(* IEC 61131-3 sources: volt/packages/volt-lsp-iec/test-corpus/lenze-mid/Device/Plc Logic/Application/Library Manager/L_MC4P_RoboticHandling (part 4) *)

(* ---- L_MC4P_TEMPLATE_FORAG.pou ---- *)
FUNCTION_BLOCK L_MC4P_TEMPLATE_FORAG
VAR
	XERROROLD : BOOL;
	WERRORIDOLD : WORD;
	XDISABLEERRORRESET : BOOL;
	XDISABLEERRORLOGGING : BOOL;
	DWERRORITFID : DWORD;
	PFBBASEAXESGROUP : POINTER TO AXES_GROUP_REF;
	PSINSTANCESTR : POINTER TO STRING;
	DISABLEERRORLOGGING : BOOL;
	DISABLEERRORRESET : BOOL;
END_VAR
END_FUNCTION_BLOCK

METHOD SETINCTANCEINFO
VAR_INPUT
	PSINSTANCENAME : POINTER TO STRING;
	ERRORITFID : DWORD;
END_VAR
END_METHOD

METHOD SETINSTANCEINFOANDAXISPOINTER
VAR_INPUT
	PAXESGROUP : POINTER TO AXES_GROUP_REF;
	PSNAME : POINTER TO STRING;
END_VAR
END_METHOD

METHOD UPDATEAXISPOINTER
VAR_INPUT
	PAXESGROUP : POINTER TO AXES_GROUP_REF;
END_VAR
END_METHOD

METHOD FB_RESETERROR
VAR_INPUT
	XERROR : BOOL;
	WERRORID : WORD;
END_VAR
END_METHOD

METHOD FB_SETERROR
VAR_INPUT
	WERRORID : L_IE1P_Error := L_IE1P_Error.NoError;
	XSETERRORSTOP : BOOL := FALSE;
END_VAR
END_METHOD

METHOD FB_SETERRORINT
VAR_INPUT
	WERRORID : L_IE1P_Error := L_IE1P_Error.NoError;
	DWINTERNALID : DWORD;
	XSETERRORSTOP : BOOL := FALSE;
END_VAR
END_METHOD

(* ---- L_MC4P_TEMPLATE_KIN.pou ---- *)
FUNCTION_BLOCK L_MC4P_TEMPLATE_KIN
VAR
	SINSTANCESTR : STRING;
	XERROROLD : BOOL;
	WERRORIDOLD : WORD;
END_VAR
END_FUNCTION_BLOCK

METHOD FB_INIT : BOOL
VAR_INPUT
	BINITRETAINS : BOOL;
	BINCOPYCODE : BOOL;
END_VAR
END_METHOD

(* ---- L_MC4P_TEMPLATE_MOVE.pou ---- *)
FUNCTION_BLOCK L_MC4P_TEMPLATE_MOVE EXTENDS L_MC4P_Template_AG_KIN
VAR
	PMOVE : POINTER TO L_MC4P_MoveContPath;
	PROFILETIME : LREAL;
	REMAININGSEGMENTLENGTH : LREAL;
	REMAININGTIMEOFPROFILE : LREAL;
	TARGETREACHED : BOOL;
	TIMEIPOACTIVE : BOOL;
END_VAR
END_FUNCTION_BLOCK

METHOD GETREMAININGSEGMENTTIME : BOOL
VAR_INPUT
	LRDISTANCETOTARGET : LREAL;
END_VAR
VAR_OUTPUT
	LRREMAININGTIME : LREAL;
END_VAR
END_METHOD

METHOD FB_INIT : BOOL
VAR_INPUT
	BINITRETAINS : BOOL;
	BINCOPYCODE : BOOL;
END_VAR
END_METHOD

(* ---- L_MC4P_TEMPLATE_MOVE_FORSMARTFBS.pou ---- *)
FUNCTION_BLOCK L_MC4P_TEMPLATE_MOVE_FORSMARTFBS EXTENDS L_MC4P_Template_Move
VAR_IN_OUT
	FBMOVE : L_MC4P_MoveContPath;
END_VAR
VAR
	PMOVE : POINTER TO L_MC4P_MoveContPath;
END_VAR
END_FUNCTION_BLOCK

(* ---- L_MC4P_TEMPLATE_MOVELICENCE.pou ---- *)
FUNCTION_BLOCK L_MC4P_TEMPLATE_MOVELICENCE EXTENDS L_MC4P_Template_Move
VAR
	LICHANDLING : L_IMHP_LLMHandling;
	MC1P_LICENCE : L_MC1P_Template_Licence_150;
END_VAR
END_FUNCTION_BLOCK

METHOD ACTIVATEAPPCREDIT : BOOL
VAR_INPUT
	XACTIVATE : BOOL;
END_VAR
END_METHOD

(* ---- L_MC4P_TEMPLATETRANSFORMATION.pou ---- *)
FUNCTION_BLOCK L_MC4P_TEMPLATETRANSFORMATION
VAR_INPUT
	PAXESGROUP : POINTER TO AXES_GROUP_KIN;
END_VAR
VAR
	IDX : INT;
	ITRAFOEXTENSION1 : L_MC4P_ITrafoExtension;
	PTRAFOEXTENSION1 : POINTER TO L_MC4P_TrafoExtensionBase;
	PTOOLTRAFO : POINTER TO L_MC4P_ToolTrafo;
	PSTORE : POINTER TO L_MC4P_IntermediateResultStore;
	PSTORE_INTERNAL : POINTER TO L_MC4P_IntermediateResultStore;
	ALRACS2JCSSCALE : ARRAY [1..6] OF LREAL := [1.0, 1.0, 1.0, 1.0, 1.0, 1.0];
	ALRJCS2ACSSCALE : ARRAY [1..6] OF LREAL := [1.0, 1.0, 1.0, 1.0, 1.0, 1.0];
END_VAR
END_FUNCTION_BLOCK

METHOD COORD2ROBOTPOS
VAR_INPUT
	PCOORD : POINTER TO ARRAY [1..6] OF LREAL;
	ECONV : L_UMTP_RotationConvention;
	ROBOTPOS : REFERENCE TO L_UMTP_RobotPos;
	XISSI : BOOL;
END_VAR
END_METHOD

METHOD TOOLTRAFOFCSTOMCSACC
VAR_INPUT
	ICOORDPROVIDER : REFERENCE TO L_MC4P_KinCoordProvider;
	BVALIDFRAME : BOOL;
	ETOOLSYSTEM : L_MC4P_ToolSystem;
END_VAR
END_METHOD

METHOD TOOLTRAFOFCSTOMCSPOS : L_MC4P_ErrorStruct
VAR_INPUT
	ICOORDPROVIDER : REFERENCE TO L_MC4P_KinCoordProvider;
	BVALIDFRAME : BOOL;
	ETOOLSYSTEM : L_MC4P_ToolSystem;
END_VAR
END_METHOD

METHOD TOOLTRAFOFCSTOMCSVEL
VAR_INPUT
	ICOORDPROVIDER : REFERENCE TO L_MC4P_KinCoordProvider;
	BVALIDFRAME : BOOL;
	ETOOLSYSTEM : L_MC4P_ToolSystem;
END_VAR
END_METHOD

METHOD TOOLTRAFOMCSTOFCSACC
VAR_INPUT
	ICOORDPROVIDER : REFERENCE TO L_MC4P_KinCoordProvider;
	BVALIDFRAME : BOOL;
	ETOOLSYSTEM : L_MC4P_ToolSystem;
END_VAR
END_METHOD

METHOD TOOLTRAFOMCSTOFCSPOS : L_MC4P_ErrorStruct
VAR_INPUT
	ICOORDPROVIDER : REFERENCE TO L_MC4P_KinCoordProvider;
	BVALIDFRAME : BOOL;
	ETOOLSYSTEM : L_MC4P_ToolSystem;
END_VAR
END_METHOD

METHOD TOOLTRAFOMCSTOFCSVEL
VAR_INPUT
	ICOORDPROVIDER : REFERENCE TO L_MC4P_KinCoordProvider;
	BVALIDFRAME : BOOL;
	ETOOLSYSTEM : L_MC4P_ToolSystem;
END_VAR
END_METHOD

METHOD TRAFOMCSTOWCSACC
VAR_INPUT
	ICOORDPROVIDER : REFERENCE TO L_MC4P_KinCoordProvider;
	BVALIDFRAME : BOOL;
END_VAR
END_METHOD

METHOD TRAFOMCSTOWCSPOS : L_MC4P_ErrorStruct
VAR_INPUT
	ICOORDPROVIDER : REFERENCE TO L_MC4P_KinCoordProvider;
	BVALIDFRAME : BOOL;
END_VAR
END_METHOD

METHOD TRAFOMCSTOWCSVEL
VAR_INPUT
	ICOORDPROVIDER : REFERENCE TO L_MC4P_KinCoordProvider;
	BVALIDFRAME : BOOL;
END_VAR
END_METHOD

METHOD TRAFOWCSTOMCSACC
VAR_INPUT
	ICOORDPROVIDER : REFERENCE TO L_MC4P_KinCoordProvider;
	BVALIDFRAME : BOOL;
END_VAR
END_METHOD

METHOD TRAFOWCSTOMCSPOS : L_MC4P_ErrorStruct
VAR_INPUT
	ICOORDPROVIDER : REFERENCE TO L_MC4P_KinCoordProvider;
	BVALIDFRAME : BOOL;
END_VAR
END_METHOD

METHOD TRAFOWCSTOMCSVEL
VAR_INPUT
	ICOORDPROVIDER : REFERENCE TO L_MC4P_KinCoordProvider;
	BVALIDFRAME : BOOL;
END_VAR
END_METHOD

METHOD CALCDINVERSEJACOBIAN : BOOL
VAR_INPUT
	ICOORDPROVIDER : L_MC4P_IKinCoordProvider;
	PDINVJACOBIAN : POINTER TO ARRAY [1..6, 1..6] OF LREAL;
END_VAR
VAR_OUTPUT
	SCERROR : L_MC4P_ErrorStruct;
END_VAR
END_METHOD

METHOD CALCDJACOBIAN : BOOL
VAR_INPUT
	ICOORDPROVIDER : L_MC4P_IKinCoordProvider;
	PDJACOBIAN : POINTER TO ARRAY [1..6, 1..6] OF LREAL;
END_VAR
VAR_OUTPUT
	SCERROR : L_MC4P_ErrorStruct;
END_VAR
END_METHOD

METHOD CALCINVERSEJACOBIAN : BOOL
VAR_INPUT
	ICOORDPROVIDER : L_MC4P_IKinCoordProvider;
	PINVJACOBIAN : POINTER TO ARRAY [1..6, 1..6] OF LREAL;
END_VAR
VAR_OUTPUT
	SCERROR : L_MC4P_ErrorStruct;
END_VAR
END_METHOD

METHOD CALCJACOBIAN : BOOL
VAR_INPUT
	ICOORDPROVIDER : L_MC4P_IKinCoordProvider;
	PJACOBIAN : POINTER TO ARRAY [1..6, 1..6] OF LREAL;
END_VAR
VAR_OUTPUT
	SCERROR : L_MC4P_ErrorStruct;
END_VAR
END_METHOD

METHOD CALCNUMERICALINVERSEJACOBIAN : L_IE1P_Error
VAR_INPUT
	ICOORDPROVIDER : L_MC4P_IKinCoordProvider;
	PINVJACOBIAN : POINTER TO ARRAY [1..6, 1..6] OF LREAL;
END_VAR
END_METHOD

METHOD CALCNUMERICALJACOBIAN : L_IE1P_Error
VAR_INPUT
	ICOORDPROVIDER : L_MC4P_IKinCoordProvider;
	PJACOBIAN : POINTER TO ARRAY [1..6, 1..6] OF LREAL;
END_VAR
END_METHOD

METHOD BWDACC : BOOL
VAR_INPUT
	ICOORDPROVIDER : REFERENCE TO L_MC4P_KinCoordProvider;
END_VAR
VAR_OUTPUT
	SCERROR : L_MC4P_ErrorStruct;
END_VAR
VAR_IN_OUT
	SCTRAFOINFO : L_MC4P_TrafoInfo;
END_VAR
END_METHOD

METHOD BWDPOS : BOOL
VAR_INPUT
	ICOORDPROVIDER : REFERENCE TO L_MC4P_KinCoordProvider;
END_VAR
VAR_OUTPUT
	SCERROR : L_MC4P_ErrorStruct;
END_VAR
VAR_IN_OUT
	SCTRAFOINFO : L_MC4P_TrafoInfo;
END_VAR
END_METHOD

METHOD BWDVEL : BOOL
VAR_INPUT
	ICOORDPROVIDER : REFERENCE TO L_MC4P_KinCoordProvider;
END_VAR
VAR_OUTPUT
	SCERROR : L_MC4P_ErrorStruct;
END_VAR
VAR_IN_OUT
	SCTRAFOINFO : L_MC4P_TrafoInfo;
END_VAR
END_METHOD

METHOD CALCPASSIVEJOINTS : L_IE1P_Error
VAR_INPUT
	PFLANGE_POS : POINTER TO ARRAY [1..6] OF LREAL;
	PJOINT_POS : POINTER TO ARRAY [1..6] OF LREAL;
	PPASSIVEJOINT_POS : POINTER TO ARRAY [1..6, 1..3] OF LREAL;
END_VAR
END_METHOD

METHOD CALCULATECONFIGURATION : L_IE1P_Error
VAR_INPUT
	PJOINT_POS : POINTER TO ARRAY [1..6] OF LREAL;
END_VAR
VAR_IN_OUT
	SCTRAFOINFO : L_MC4P_TrafoInfo;
END_VAR
END_METHOD

METHOD FWDACC : BOOL
VAR_INPUT
	ICOORDPROVIDER : REFERENCE TO L_MC4P_KinCoordProvider;
END_VAR
VAR_OUTPUT
	SCERROR : L_MC4P_ErrorStruct;
END_VAR
VAR_IN_OUT
	SCTRAFOINFO : L_MC4P_TrafoInfo;
END_VAR
END_METHOD

METHOD FWDPOS : BOOL
VAR_INPUT
	ICOORDPROVIDER : REFERENCE TO L_MC4P_KinCoordProvider;
END_VAR
VAR_OUTPUT
	SCERROR : L_MC4P_ErrorStruct;
END_VAR
VAR_IN_OUT
	SCTRAFOINFO : L_MC4P_TrafoInfo;
END_VAR
END_METHOD

METHOD FWDVEL : BOOL
VAR_INPUT
	ICOORDPROVIDER : REFERENCE TO L_MC4P_KinCoordProvider;
END_VAR
VAR_OUTPUT
	SCERROR : L_MC4P_ErrorStruct;
END_VAR
VAR_IN_OUT
	SCTRAFOINFO : L_MC4P_TrafoInfo;
END_VAR
END_METHOD

METHOD GETTRAFOEXTENSION1 : L_MC4P_ITrafoExtension
VAR_OUTPUT
	PFB : POINTER TO L_MC4P_TrafoExtensionBase;
END_VAR
END_METHOD

METHOD MCS_ORIENTATIONCHECK : L_IE1P_Error
VAR_IN_OUT
	ICOORDPROVIDER : L_MC4P_KinCoordProvider;
END_VAR
END_METHOD

METHOD SETTRAFOEXTENSION1
VAR_INPUT
	TRAFOEXTENSION : L_MC4P_ITrafoExtension;
	PFB : POINTER TO L_MC4P_TrafoExtensionBase;
END_VAR
END_METHOD

METHOD CHECKNEIGHBOURHOOD : L_IE1P_Error
VAR_INPUT
	PJOINT_POS : POINTER TO ARRAY [1..6] OF LREAL;
END_VAR
VAR_IN_OUT
	SCTRAFOINFO : L_MC4P_TrafoInfo;
END_VAR
END_METHOD

METHOD COUNTREVOLUTIONSFORWARDTRAFO : L_IE1P_Error
VAR_INPUT
	PJOINT_POS : POINTER TO ARRAY [1..6] OF LREAL;
END_VAR
VAR_IN_OUT
	SCTRAFOINFO : L_MC4P_TrafoInfo;
END_VAR
END_METHOD

METHOD IDENTIFYTRAFOCASE : L_IE1P_Error
VAR_INPUT
	PKART_POS : POINTER TO ARRAY [1..6] OF LREAL;
	PMCS_POS : POINTER TO ARRAY [1..6] OF LREAL;
	PFLANGE_POS : POINTER TO ARRAY [1..6] OF LREAL;
	PJOINT_POS : POINTER TO ARRAY [1..6] OF LREAL;
	PAXES_POS : POINTER TO ARRAY [1..6] OF LREAL;
END_VAR
VAR_IN_OUT
	ILOWERSYSTEM : INT;
	IUPPERSYSTEM : INT;
END_VAR
END_METHOD

METHOD PRELOADCONSTANTAXES
VAR_INPUT
	PACSPOS : POINTER TO ARRAY [1..6] OF LREAL;
	PJCSPOS : POINTER TO ARRAY [1..6] OF LREAL;
	PFCSPOS : POINTER TO ARRAY [1..6] OF LREAL;
	PMCSPOS : POINTER TO ARRAY [1..6] OF LREAL;
	PWCSPOS : POINTER TO ARRAY [1..6] OF LREAL;
END_VAR
VAR_IN_OUT
	SCTRAFOINFO : L_MC4P_TrafoInfo;
END_VAR
END_METHOD

METHOD ADDTURNSTOJOINTS : L_IE1P_Error
VAR_INPUT
	PFLANGE_POS : POINTER TO ARRAY [1..6] OF LREAL;
	PJOINT_POS : POINTER TO ARRAY [1..6] OF LREAL;
END_VAR
VAR_IN_OUT
	SCTRAFOINFO : L_MC4P_TrafoInfo;
END_VAR
END_METHOD

METHOD CALCBACKWARDTRANSFORMATIONACC : L_IE1P_Error
VAR_INPUT
	PSTORE : POINTER TO L_MC4P_IntermediateResultStore;
END_VAR
VAR_IN_OUT
	SCTRAFOINFO : L_MC4P_TrafoInfo;
END_VAR
END_METHOD

METHOD CALCBACKWARDTRANSFORMATIONPOS : L_IE1P_Error
VAR_INPUT
	PSTORE : POINTER TO L_MC4P_IntermediateResultStore;
END_VAR
VAR_IN_OUT
	SCTRAFOINFO : L_MC4P_TrafoInfo;
END_VAR
END_METHOD

METHOD CALCBACKWARDTRANSFORMATIONVEL : L_IE1P_Error
VAR_INPUT
	PSTORE : POINTER TO L_MC4P_IntermediateResultStore;
END_VAR
VAR_IN_OUT
	SCTRAFOINFO : L_MC4P_TrafoInfo;
END_VAR
END_METHOD

METHOD CALCFORWARDTRANSFORMATIONACC : L_IE1P_Error
VAR_INPUT
	PSTORE : POINTER TO L_MC4P_IntermediateResultStore;
END_VAR
VAR_IN_OUT
	SCTRAFOINFO : L_MC4P_TrafoInfo;
END_VAR
END_METHOD

METHOD CALCFORWARDTRANSFORMATIONPOS : L_IE1P_Error
VAR_INPUT
	PSTORE : POINTER TO L_MC4P_IntermediateResultStore;
END_VAR
VAR_IN_OUT
	SCTRAFOINFO : L_MC4P_TrafoInfo;
END_VAR
END_METHOD

METHOD CALCFORWARDTRANSFORMATIONVEL : L_IE1P_Error
VAR_INPUT
	PSTORE : POINTER TO L_MC4P_IntermediateResultStore;
END_VAR
VAR_IN_OUT
	SCTRAFOINFO : L_MC4P_TrafoInfo;
END_VAR
END_METHOD

METHOD CALCPASSIVEJOINTSACC : L_IE1P_Error
VAR_INPUT
	PSTORE : POINTER TO L_MC4P_IntermediateResultStore;
END_VAR
VAR_IN_OUT
	SCTRAFOINFO : L_MC4P_TrafoInfo;
END_VAR
END_METHOD

METHOD CALCPASSIVEJOINTSPOS : L_IE1P_Error
VAR_INPUT
	PSTORE : POINTER TO L_MC4P_IntermediateResultStore;
END_VAR
VAR_IN_OUT
	SCTRAFOINFO : L_MC4P_TrafoInfo;
END_VAR
END_METHOD

METHOD CALCPASSIVEJOINTSVEL : L_IE1P_Error
VAR_INPUT
	PSTORE : POINTER TO L_MC4P_IntermediateResultStore;
END_VAR
VAR_IN_OUT
	SCTRAFOINFO : L_MC4P_TrafoInfo;
END_VAR
END_METHOD

METHOD FINALIZEBWD : L_IE1P_Error
VAR_IN_OUT
	SCTRAFOINFO : L_MC4P_TrafoInfo;
	ICOORDPROVIDER : L_MC4P_KinCoordProvider;
END_VAR
END_METHOD

METHOD TRANSFORMREVOLUTEJOINTS : L_IE1P_Error
VAR_INPUT
	PJCSPOS : POINTER TO ARRAY [1..6] OF LREAL;
END_VAR
VAR_IN_OUT
	SCTRAFOINFO : L_MC4P_TrafoInfo;
END_VAR
END_METHOD

(* ---- L_MC4P_TOOLCONTROL.pou ---- *)
FUNCTION_BLOCK L_MC4P_TOOLCONTROL
VAR_INPUT
	XENABLE : BOOL;
	ETOOLSYSTEM : L_MC4P_ToolSystem;
END_VAR
VAR_OUTPUT
	XBUSY : BOOL;
	XERROR : BOOL;
	EERRORID : L_IE1P_Error;
	XPULSEON : BOOL;
	XPULSEOFF : BOOL;
	LRTIMETOPULSE : LREAL;
END_VAR
VAR_IN_OUT
	AXESGROUP : AXES_GROUP_KIN;
END_VAR
VAR
	_ON_TRIG : R_Trig;
	_OFF_TRIG : R_Trig;
	_ITFTOOL : L_MC4P_IToolInfo;
	_NSTATE : DWORD := 10;
	_ETOOLSYSTEMFREEZE : L_MC4P_ToolSystem;
	_PTOOL : POINTER TO L_MC4P_ToolTrafo;
	_ETOOLREQU : L_MC4P_ToolRequest;
	_LRSWITCHTIME : LREAL;
	_MODEL : L_UBUP_BehaviourModel_LCon;
END_VAR
END_FUNCTION_BLOCK

METHOD CYCLICACTION
VAR_INPUT
	ITFTIMINGCONTROLLER : L_UBUP.L_UBUP_ITimingController;
END_VAR
VAR_OUTPUT
	XCOMPLETE : BOOL;
	XABORT : BOOL;
	IERRORID : INT;
END_VAR
END_METHOD

METHOD FINALIZEACTION
VAR_INPUT
	XABORTPROPOSED : BOOL;
	IERRORIDPROPOSED : INT;
END_VAR
VAR_OUTPUT
	XCOMPLETE : BOOL;
	XABORT : BOOL;
	IERRORID : INT;
END_VAR
END_METHOD

METHOD RESETACTION
VAR_OUTPUT
	XCOMPLETE : BOOL;
END_VAR
END_METHOD

METHOD STARTACTION
VAR_OUTPUT
	XCOMPLETE : BOOL;
	IERRORID : INT;
END_VAR
END_METHOD

(* ---- L_MC4P_TOOLTRAFO.pou ---- *)
FUNCTION_BLOCK L_MC4P_TOOLTRAFO
VAR_INPUT
	TOOLPARAM : L_MC4P_TOOL_REF;
	EROTATIONCONVENTION : L_UMTP_RotationConvention;
	ISWITCHONTIME : INT;
	ISWITCHOFFTIME : INT;
END_VAR
VAR_OUTPUT
	T_01 : ARRAY [1..4, 1..4] OF LREAL;
	T_01_FRAME : L_UMTP_RobotFrame;
	T_10 : ARRAY [1..4, 1..4] OF LREAL;
	T_10_FRAME : L_UMTP_RobotFrame;
END_VAR
VAR
	TOOLPARAMINT : L_MC4P_TOOL_REF;
	EROTATIONCONVENTIONINT : L_UMTP_RotationConvention;
	PAXESGROUP : POINTER TO AXES_GROUP_KIN;
END_VAR
END_FUNCTION_BLOCK

METHOD CALCHOMTRAFO
VAR_IN_OUT
	AXESGROUP : AXES_GROUP_KIN;
END_VAR
END_METHOD

METHOD ROTATE_FCS2TCS
VAR_INPUT
	PALRIN : POINTER TO ARRAY [1..6] OF LREAL;
	PALROUT : POINTER TO ARRAY [1..6] OF LREAL;
END_VAR
END_METHOD

METHOD ROTATE_TCS2FCS
VAR_INPUT
	PALRIN : POINTER TO ARRAY [1..6] OF LREAL;
	PALROUT : POINTER TO ARRAY [1..6] OF LREAL;
END_VAR
END_METHOD

(* ---- L_MC4P_TRACELIST.pou ---- *)
FUNCTION_BLOCK L_MC4P_TRACELIST
VAR_INPUT
	XENABLE : BOOL;
	PAXESGROUP : POINTER TO AXES_GROUP_KIN;
END_VAR
VAR
	PLISTELEMENT : POINTER TO L_MC4P_ListElement;
	VISULISTTABLE : ARRAY [0..L_MC4P_Constants.SizeVisuArray] OF L_MC4P_VisuListTableData;
	BFINISHED : BOOL := 0;
	IINDEX : INT := 0;
	XREADFROMLISTELEMENTLAST : BOOL := TRUE;
	HEVENTCOMMCYCLE : Systypes.RTS_IEC_HANDLE := SysTypes.RTS_INVALID_HANDLE;
	HINTERFACECOMMCYCLE : Systypes.RTS_IEC_HANDLE := SysTypes.RTS_INVALID_HANDLE;
	ITFCALLBACK : CmpEventMgr.ICmpEventCallback;
	DWEVENTCOUNTER : DWORD;
END_VAR
END_FUNCTION_BLOCK

METHOD FILLVISULISTTABLEELEMENT
END_METHOD

METHOD MAIN
END_METHOD

METHOD EVENTCALLBACK : UDINT
VAR_INPUT
	PEVENTPARAM : POINTER TO EventParam;
END_VAR
END_METHOD

METHOD REGISTEREVENT
END_METHOD

METHOD UNREGISTEREVENT
END_METHOD

(* ---- L_MC4P_TRACKCONVEYORBELT_INTERNAL.pou ---- *)
FUNCTION_BLOCK L_MC4P_TRACKCONVEYORBELT_INTERNAL EXTENDS L_MC4P_TrackKinematics
VAR_INPUT
	ITFCONVEYORBELT : L_MC1P_IAXIS_REF_MASTERVALUES;
	EXECUTE : BOOL;
	ABORT : BOOL;
	CONVEYORBELTORIGIN : ARRAY [1..6] OF LREAL;
	INITIALOBJECTPOSITION : ARRAY [1..6] OF LREAL;
	COORDSYSTEM : L_MC4P_CoordSystem;
	COORDTYPE : L_MC4P_CoordType;
	CLUTCHDISTANCE : LREAL;
	CLUTCHTIME : LREAL;
	CLUTCHTIMEABORT : LREAL;
	SETDYNPCS : BOOL := TRUE;
END_VAR
VAR_OUTPUT
	DONE : BOOL;
	BUSY : BOOL;
	ACTIVE : BOOL;
	COMMANDABORTED : BOOL;
	ERROR : BOOL;
	ERRORID : L_IE1P_Error;
	INSYNC : BOOL;
	DYNAMICPCSSET : BOOL;
END_VAR
VAR
	LRCONVBELTPOSITIONOLD : LREAL := 0;
	LRCOUNTEDMODULOCYCLES : LREAL := 0;
	EMASTERDIRECTIONSAVED : MC_Direction := MC_Direction.mcPositiveDirection;
	XMASTERVALID : BOOL;
	FBCONSIDERCVUNSTEADY : L_MC1P_ConsiderMasterUnsteady;
	CLUTCHEXTERNAL : LREAL;
END_VAR
END_FUNCTION_BLOCK

METHOD GETCLUTCHPARAMETER : BOOL
VAR_OUTPUT
	EERRORID : L_IE1P_Error;
END_VAR
END_METHOD

METHOD GETINITOBJPOS : MC_Coord_Ref
END_METHOD

METHOD GETMASTERDIRECTION : BOOL
VAR_INPUT
	ITFCONVEYORBELT : L_MC1P_IAXIS_REF_MASTERVALUES;
END_VAR
END_METHOD

METHOD GETMASTERVALUES : BOOL
VAR_INPUT
	PALRINITMASTERPOS : POINTER TO ARRAY [1..6] OF LREAL;
	PASCCNVVALUESCCS : POINTER TO ARRAY [1..6] OF L_MC4P_AxisProfile;
	PASCCNVVALUESCCSOLD : POINTER TO ARRAY [1..6] OF L_MC4P_AxisProfile;
	LRMASTERPOSEXTRAPOL : LREAL;
END_VAR
END_METHOD

METHOD MAIN
VAR_INPUT
	ITFCONVEYORBELT : L_MC1P_IAXIS_REF_MASTERVALUES;
END_VAR
VAR_IN_OUT
	AXESGROUP : AXES_GROUP_KIN;
	FBBASE : L_MC4P_Template_AG_KIN;
END_VAR
END_METHOD

METHOD PARAMETERFREEZE
VAR_OUTPUT
	EERRORID : L_IE1P_Error;
END_VAR
VAR_IN_OUT
	AXESGROUP : AXES_GROUP_KIN;
	FBBASE : L_MC4P_Template_AG_KIN;
END_VAR
END_METHOD

METHOD SYNCINONPOS : BOOL
VAR_INPUT
	PASCCNVVALUESCCS : POINTER TO ARRAY [1..6] OF L_MC4P_AxisProfile;
	ALRSUPERPOSPOSATCLUTCH : ARRAY [1..3] OF LREAL;
	PTRAFO_BASE_MCS : POINTER TO L_MC4P_CoordTrafo;
	LRCLUTCHDISTANCE : LREAL;
END_VAR
VAR_OUTPUT
	XINSYNC : BOOL;
END_VAR
VAR_IN_OUT
	AXESGROUP : AXES_GROUP_KIN;
	FBBASE : L_MC4P_Template_AG_KIN;
END_VAR
END_METHOD

METHOD SYNCINONTIME : BOOL
VAR_INPUT
	PASCCNVVALUESCCS : POINTER TO ARRAY [1..6] OF L_MC4P_AxisProfile;
	ALRSUPERPOSPOSATCLUTCH : ARRAY [1..3] OF LREAL;
	PTRAFO_BASE_MCS : POINTER TO L_MC4P_CoordTrafo;
	LRCLUTCHDISTANCE : LREAL;
END_VAR
VAR_OUTPUT
	XINSYNC : BOOL;
END_VAR
VAR_IN_OUT
	AXESGROUP : AXES_GROUP_KIN;
	FBBASE : L_MC4P_Template_AG_KIN;
END_VAR
END_METHOD

METHOD SYNCOUTONPOS : BOOL
VAR_INPUT
	PASCCNVVALUESCCS : POINTER TO ARRAY [1..6] OF L_MC4P_AxisProfile;
	ALRSUPERPOSPOSATCLUTCH : ARRAY [1..3] OF LREAL;
	PTRAFO_BASE_MCS : POINTER TO L_MC4P_CoordTrafo;
	LRCLUTCHDISTANCE : LREAL;
END_VAR
VAR_OUTPUT
	XSYNCOUTDONE : BOOL;
END_VAR
VAR_IN_OUT
	AXESGROUP : AXES_GROUP_KIN;
	FBBASE : L_MC4P_Template_AG_KIN;
END_VAR
END_METHOD

METHOD SYNCOUTONTIME : BOOL
VAR_INPUT
	PASCCNVVALUESCCS : POINTER TO ARRAY [1..6] OF L_MC4P_AxisProfile;
	ALRSUPERPOSPOSATCLUTCH : ARRAY [1..3] OF LREAL;
	PTRAFO_BASE_MCS : POINTER TO L_MC4P_CoordTrafo;
	LRCLUTCHDISTANCE : LREAL;
	XSYNCOUTKEEPPOSITION : BOOL;
END_VAR
VAR_OUTPUT
	XSYNCOUTDONE : BOOL;
END_VAR
VAR_IN_OUT
	AXESGROUP : AXES_GROUP_KIN;
	FBBASE : L_MC4P_Template_AG_KIN;
END_VAR
END_METHOD

METHOD SYNCHRON : BOOL
VAR_INPUT
	PASCCNVVALUESCCS : POINTER TO ARRAY [1..6] OF L_MC4P_AxisProfile;
	PTRAFO_BASE_MCS : POINTER TO L_MC4P_CoordTrafo;
END_VAR
END_METHOD

(* ---- L_MC4P_TRACKKINEMATICS.pou ---- *)
FUNCTION_BLOCK L_MC4P_TRACKKINEMATICS
VAR_INPUT
	EMASTERVALUESOURCE : MC_SOURCE := MC_SOURCE.mcCommandedValue;
END_VAR
VAR
	XDONE_INTERN : BOOL;
	XBUSY_INTERN : BOOL;
	XACTIVE_INTERN : BOOL;
	XCOMMANDABORTED_INTERN : BOOL;
	XERROR_INTERN : BOOL;
	EERRORID_INTERN : L_IE1P_Error;
	XINSYNC_INTERN : BOOL;
	DYNAMICPCSSET_INTERN : BOOL;
	WSTEP : L_MC4P_TrackKinematicsStates;
	WSTEPOLD : L_MC4P_TrackKinematicsStates;
	XEXECUTEOLD : BOOL;
	XSETDYNPCSINDEPENDANTOLD : BOOL;
	XCALCDYNPCS : BOOL;
	XERRORLASTCYCLE : BOOL;
	XABORTOLD : BOOL;
	XABORTEDMOVEMENT : BOOL;
	XABORTFB : BOOL;
	XRESTARTSYNC : BOOL;
	XWINSTANCE : __XWORD;
	SCINPUTPARAM : L_MC4P_TrackInputParam;
	PSCSUPERPOSDATA : POINTER TO L_MC4P_SuperposHandler;
	SCINITIALPCSINTERN : L_MC4P_CoordTrafo;
	PSCHANDSHAKE : POINTER TO L_MC4P_TrackingHandshake;
	ASCCONVEYORVALUES : ARRAY [1..6] OF L_MC4P_AxisProfile;
	ASCCONVEYORVALUESFIXED : ARRAY [1..6] OF L_MC4P_AxisProfile;
	ASCCONVEYORVALUESOLD : ARRAY [1..6] OF L_MC4P_AxisProfile;
	XCLUTCHINITDONE : BOOL;
	ASCENDSLAVE : ARRAY [1..7] OF L_MC4P_AxisProfile;
	ASCSTARTSLAVE : ARRAY [1..7] OF L_MC4P_AxisProfile;
	ALRMASTERCLUTCHPOS : ARRAY [1..6] OF LREAL;
	ACLUTCHFB : ARRAY [1..7] OF L_MC4P_Clutch;
	ALRCNVPOSATCLINCCS : ARRAY [1..6] OF LREAL;
	ALRSUPERPOSPOSTEMP : ARRAY [1..3] OF LREAL;
	LRTIMECOUNTER : LREAL;
	LRCLUTCHTIMEABORTDEFAULT : LREAL := 1.0;
	LRCLUTCHEXTERNAL : LREAL := -1.0;
	XUSECLUTCHEXTERNAL : BOOL;
	ASCSLAVEEXTRAPOL : ARRAY [1..7] OF L_MC4P_AxisProfile;
	ALRACCMINUS0 : ARRAY [1..7] OF LREAL;
	ALRVELMINUS0 : ARRAY [1..7] OF LREAL;
	ALRVELMINUS1 : ARRAY [1..7] OF LREAL;
	ALRPOSMINUS0 : ARRAY [1..7] OF LREAL;
	ALRPOSMINUS1 : ARRAY [1..7] OF LREAL;
	ALRPOSMINUS2 : ARRAY [1..7] OF LREAL;
	XABORTAGSTOPPING : BOOL;
	XSTATEMACHINE : BOOL;
	MASTERVALUESOURCE : MC_SOURCE;
END_VAR
END_FUNCTION_BLOCK

METHOD CALCDYNPCS : BOOL
VAR_INPUT
	BINITIALCALL : BOOL;
	PASCACTCNVVALUESCCS : POINTER TO ARRAY [1..6] OF L_MC4P_AxisProfile;
END_VAR
VAR_IN_OUT
	AXESGROUP : AXES_GROUP_KIN;
	FBBASE : L_MC4P_Template_AG_KIN;
END_VAR
END_METHOD

METHOD FB_INIT : BOOL
VAR_INPUT
	BINITRETAINS : BOOL;
	BINCOPYCODE : BOOL;
END_VAR
END_METHOD

METHOD GETCLUTCHPARAMETER : BOOL
VAR_OUTPUT
	EERRORID : L_IE1P_Error;
END_VAR
END_METHOD

METHOD GETINITOBJPOS : MC_Coord_Ref
END_METHOD

METHOD GETMASTERVALUES : BOOL
VAR_INPUT
	PALRINITMASTERPOS : POINTER TO ARRAY [1..6] OF LREAL;
	PASCCNVVALUESCCS : POINTER TO ARRAY [1..6] OF L_MC4P_AxisProfile;
	PASCCNVVALUESCCSOLD : POINTER TO ARRAY [1..6] OF L_MC4P_AxisProfile;
	LRMASTERPOSEXTRAPOL : LREAL;
END_VAR
END_METHOD

METHOD PARAMETERFREEZE
VAR_OUTPUT
	EERRORID : L_IE1P_Error;
END_VAR
VAR_IN_OUT
	AXESGROUP : AXES_GROUP_KIN;
	FBBASE : L_MC4P_Template_AG_KIN;
END_VAR
END_METHOD

METHOD PASSTHROUGHTRACKINGOFFSETRESET : BOOL
VAR_IN_OUT
	AXESGROUP : AXES_GROUP_KIN;
	FBBASE : L_MC4P_Template_AG_KIN;
END_VAR
END_METHOD

METHOD RESETSUPERPOSCLUTCHINITDONE
END_METHOD

METHOD SETCONVEYORVALUESFIXED
END_METHOD

METHOD SYNCINONPOS : BOOL
VAR_INPUT
	PASCCNVVALUESCCS : POINTER TO ARRAY [1..6] OF L_MC4P_AxisProfile;
	ALRSUPERPOSPOSATCLUTCH : ARRAY [1..3] OF LREAL;
	PTRAFO_BASE_MCS : POINTER TO L_MC4P_CoordTrafo;
	LRCLUTCHDISTANCE : LREAL;
END_VAR
VAR_OUTPUT
	XINSYNC : BOOL;
END_VAR
VAR_IN_OUT
	AXESGROUP : AXES_GROUP_KIN;
	FBBASE : L_MC4P_Template_AG_KIN;
END_VAR
END_METHOD

METHOD SYNCINONTIME : BOOL
VAR_INPUT
	PASCCNVVALUESCCS : POINTER TO ARRAY [1..6] OF L_MC4P_AxisProfile;
	ALRSUPERPOSPOSATCLUTCH : ARRAY [1..3] OF LREAL;
	PTRAFO_BASE_MCS : POINTER TO L_MC4P_CoordTrafo;
	LRCLUTCHDISTANCE : LREAL;
END_VAR
VAR_OUTPUT
	XINSYNC : BOOL;
END_VAR
VAR_IN_OUT
	AXESGROUP : AXES_GROUP_KIN;
	FBBASE : L_MC4P_Template_AG_KIN;
END_VAR
END_METHOD

METHOD SYNCOUTONPOS : BOOL
VAR_INPUT
	PASCCNVVALUESCCS : POINTER TO ARRAY [1..6] OF L_MC4P_AxisProfile;
	ALRSUPERPOSPOSATCLUTCH : ARRAY [1..3] OF LREAL;
	PTRAFO_BASE_MCS : POINTER TO L_MC4P_CoordTrafo;
	LRCLUTCHDISTANCE : LREAL;
END_VAR
VAR_OUTPUT
	XSYNCOUTDONE : BOOL;
END_VAR
VAR_IN_OUT
	AXESGROUP : AXES_GROUP_KIN;
	FBBASE : L_MC4P_Template_AG_KIN;
END_VAR
END_METHOD

METHOD SYNCOUTONTIME : BOOL
VAR_INPUT
	PASCCNVVALUESCCS : POINTER TO ARRAY [1..6] OF L_MC4P_AxisProfile;
	ALRSUPERPOSPOSATCLUTCH : ARRAY [1..3] OF LREAL;
	PTRAFO_BASE_MCS : POINTER TO L_MC4P_CoordTrafo;
	LRCLUTCHDISTANCE : LREAL;
	XSYNCOUTKEEPPOSITION : BOOL;
END_VAR
VAR_OUTPUT
	XSYNCOUTDONE : BOOL;
END_VAR
VAR_IN_OUT
	AXESGROUP : AXES_GROUP_KIN;
	FBBASE : L_MC4P_Template_AG_KIN;
END_VAR
END_METHOD

METHOD SYNCHRON : BOOL
VAR_INPUT
	PASCCNVVALUESCCS : POINTER TO ARRAY [1..6] OF L_MC4P_AxisProfile;
	PTRAFO_BASE_MCS : POINTER TO L_MC4P_CoordTrafo;
END_VAR
END_METHOD

METHOD STATE_AGSTOP
VAR_INPUT
	XEXECUTE : BOOL;
END_VAR
VAR_IN_OUT
	AXESGROUP : AXES_GROUP_KIN;
	FBBASE : L_MC4P_Template_AG_KIN;
END_VAR
END_METHOD

METHOD STATE_ABORTING
VAR_INPUT
	XEXECUTE : BOOL;
END_VAR
VAR_IN_OUT
	AXESGROUP : AXES_GROUP_KIN;
	FBBASE : L_MC4P_Template_AG_KIN;
END_VAR
END_METHOD

METHOD STATE_ERROR
VAR_INPUT
	XEXECUTE : BOOL;
END_VAR
VAR_IN_OUT
	AXESGROUP : AXES_GROUP_KIN;
	FBBASE : L_MC4P_Template_AG_KIN;
END_VAR
END_METHOD

METHOD STATE_INITIAL
VAR_INPUT
	XEXECUTE : BOOL;
	XSETDYNPCSINDEPENDANT : BOOL;
END_VAR
VAR_IN_OUT
	AXESGROUP : AXES_GROUP_KIN;
	FBBASE : L_MC4P_Template_AG_KIN;
END_VAR
END_METHOD

METHOD STATE_SYNCIN
VAR_INPUT
	XEXECUTE : BOOL;
END_VAR
VAR_IN_OUT
	AXESGROUP : AXES_GROUP_KIN;
	FBBASE : L_MC4P_Template_AG_KIN;
END_VAR
END_METHOD

METHOD STATE_SYNCOUT
VAR_INPUT
	XEXECUTE : BOOL;
	XABORT : BOOL;
END_VAR
VAR_IN_OUT
	AXESGROUP : AXES_GROUP_KIN;
	FBBASE : L_MC4P_Template_AG_KIN;
END_VAR
END_METHOD

METHOD STATE_SYNCHRON
VAR_INPUT
	XEXECUTE : BOOL;
END_VAR
VAR_IN_OUT
	AXESGROUP : AXES_GROUP_KIN;
	FBBASE : L_MC4P_Template_AG_KIN;
END_VAR
END_METHOD

METHOD STATE_WAITFORMOTION
VAR_INPUT
	XEXECUTE : BOOL;
END_VAR
VAR_IN_OUT
	AXESGROUP : AXES_GROUP_KIN;
	FBBASE : L_MC4P_Template_AG_KIN;
END_VAR
END_METHOD

METHOD TRACKKINEMATICS
VAR_INPUT
	XEXECUTE : BOOL;
	XABORT : BOOL;
	XSETDYNPCSINDEPENDANT : BOOL;
END_VAR
VAR_IN_OUT
	AXESGROUP : AXES_GROUP_KIN;
	FBBASE : L_MC4P_Template_AG_KIN;
END_VAR
END_METHOD

(* ---- L_MC4P_TRAFOEXTENSIONBASE.pou ---- *)
FUNCTION_BLOCK L_MC4P_TRAFOEXTENSIONBASE EXTENDS L_MC4P_Template_AG_KIN
END_FUNCTION_BLOCK

METHOD BACKWARDTRANSFORMATIONEXTENSION : L_IE1P_Error
VAR_INPUT
	PAXES_POS : POINTER TO ARRAY [1..6] OF LREAL;
	PJOINT_POS : POINTER TO ARRAY [1..6] OF LREAL;
END_VAR
END_METHOD

METHOD CHECKINPUTS : L_IE1P_Error
VAR_IN_OUT
	AXESGROUP : AXES_GROUP_KIN;
END_VAR
END_METHOD

METHOD FORWARDTRANSFORMATIONEXTENSION : L_IE1P_Error
VAR_INPUT
	PAXES_POS : POINTER TO ARRAY [1..6] OF LREAL;
	PJOINT_POS : POINTER TO ARRAY [1..6] OF LREAL;
END_VAR
END_METHOD

METHOD GENERALIZEDFORCE_ACS2JCS : L_IE1P_Error
VAR_INPUT
	PAXES_FORCE : POINTER TO ARRAY [1..6] OF LREAL;
	PJOINT_FORCE : POINTER TO ARRAY [1..6] OF LREAL;
END_VAR
END_METHOD

METHOD GENERALIZEDFORCE_JCS2ACS : L_IE1P_Error
VAR_INPUT
	PAXES_FORCE : POINTER TO ARRAY [1..6] OF LREAL;
	PJOINT_FORCE : POINTER TO ARRAY [1..6] OF LREAL;
END_VAR
END_METHOD

(* ---- L_MC4P_TRAFOINFO.pou ---- *)
FUNCTION_BLOCK L_MC4P_TRAFOINFO
VAR_INPUT
	ALITURNS : ARRAY [1..6] OF LINT;
	AIQUADRANT : ARRAY [1..6] OF INT;
	AICONFIG : ARRAY [1..6] OF INT;
	XCHECKQUADRANT : BOOL;
	ALRNEIGHBOUR : ARRAY [1..6] OF LREAL;
	ICHECKNEIGHBOURHOOD : INT;
	ETOOLSYSTEM : L_MC4P_ToolSystem;
END_VAR
VAR
	TYPEID : L_MC4P_KinematicType;
END_VAR
END_FUNCTION_BLOCK

METHOD COPYFROM : L_IE1P_Error
VAR_INPUT
	SCSOURCE : REFERENCE TO L_MC4P_TrafoInfo;
END_VAR
END_METHOD

METHOD FB_INIT : BOOL
VAR_INPUT
	BINITRETAINS : BOOL;
	BINCOPYCODE : BOOL;
END_VAR
END_METHOD

METHOD RESET
END_METHOD

(* ---- L_MC4P_VIRTUALTIME.pou ---- *)
FUNCTION_BLOCK L_MC4P_VIRTUALTIME
VAR_INPUT
	XENABLE : BOOL;
	LRCYCLETIME : LREAL;
	LROVRREQUESTED : LREAL := 1.0;
END_VAR
VAR_OUTPUT
	LRVIRTUALTIMECYCLE : LREAL;
	LROVRACTUAL : LREAL;
	LRDOVRACTUAL : LREAL;
	XERROR : BOOL := FALSE;
	EERRORID : L_IE1P_Error;
END_VAR
VAR
	_REFTIMEFILTER : REFERENCE TO L_USPP_Filter;
	_FBPT2 : L_USPP_PT2Filter;
	_XTIMEFILTERDONE : BOOL;
	_XPAUSE : BOOL := FALSE;
	_XFORCEOVREQ1 : BOOL := FALSE;
	XPAUSE : BOOL;
END_VAR
END_FUNCTION_BLOCK

METHOD CALLTIMEFILTER
END_METHOD

METHOD ENTRYCYCLE
END_METHOD

METHOD FORCESTOPOVREQ1
END_METHOD

METHOD IDENTIFYTIMEFILTER : BOOL
VAR_INPUT
	FBTIMEFILTER : REFERENCE TO L_USPP_Filter;
END_VAR
END_METHOD

METHOD LEAVECYCLE
END_METHOD

METHOD REPLACETIMEFILTER
VAR_INPUT
	FBTIMEFILTER : REFERENCE TO L_USPP_Filter;
END_VAR
END_METHOD

METHOD FB_INIT : BOOL
VAR_INPUT
	BINITRETAINS : BOOL;
	BINCOPYCODE : BOOL;
END_VAR
END_METHOD

(* ---- L_MC4P_VISU_AXES_GROUP_KIN.pou ---- *)
FUNCTION_BLOCK L_MC4P_VISU_AXES_GROUP_KIN
VAR_INPUT
	M_INPUT_INST_STR : STRING;
	XENABLEVISU : BOOL := FALSE;
	XTEST : BOOL := FALSE;
	XSHOWPATH : BOOL := TRUE;
	PAXESGROUP : POINTER TO AXES_GROUP_KIN;
END_VAR
VAR
	FBKINCOORDPROVIDER : L_MC4P_KinCoordProvider;
	XENABLEVISUOLD : BOOL := FALSE;
	ALRACSTESTPOS : ARRAY [1..6] OF LREAL := [6(0)];
	ALRACSPOS : ARRAY [1..6] OF LREAL := [6(0)];
	ALRJCSPOS : ARRAY [1..6] OF LREAL := [6(0)];
	ALRXTCS_MCS : ARRAY [1..6] OF LREAL := [6(0)];
	ALRXTCS_WCS : ARRAY [1..6] OF LREAL := [6(0)];
	ALRXEE_MCS : ARRAY [1..6] OF LREAL := [6(0)];
	ALRMCS_WCS : ARRAY [1..6] OF LREAL := [6(0)];
	ALRWCS_MCS : ARRAY [1..6] OF LREAL := [6(0)];
	COORDTMP : MC_COORD_REF;
	AXDISPLAYINVISIBLE : ARRAY [1..12] OF BOOL;
	AXDISPLAYINACTIVE : ARRAY [1..12] OF BOOL;
	XSHOWCONFIGELEMENTS : BOOL := FALSE;
	IDX : INT;
	XINIT : BOOL := TRUE;
	XREINIT : BOOL := TRUE;
	EKINEMATIC : L_MC4P_KinematicType := L_MC4P_KinematicType.NoKinematic;
	XSCALING : BOOL;
	FRAMELIMITATION : ARRAY [1..6] OF LREAL;
	XSHOWFRAME : BOOL := FALSE;
	XRECALCSCALINGS : BOOL := FALSE;
	XVISUPCSACTIVE : BOOL := FALSE;
	LRUNITSTOPIXELFRAME1 : LREAL := 1;
	LRUNITSTOPIXELFRAME2 : LREAL := 1;
	LRMCS0FRAME1 : ARRAY [1..2] OF LREAL := [200, 200];
	LRMCS0FRAME2 : ARRAY [1..2] OF LREAL := [50, 350];
	ALRRTCS2MCS : ARRAY [1..3, 1..3] OF LREAL;
	ALRRMCS2TCS : ARRAY [1..3, 1..3] OF LREAL;
	ALRRMCS2FRAME1 : ARRAY [1..3, 1..3] OF LREAL;
	ALRRFRAME12MCS : ARRAY [1..3, 1..3] OF LREAL;
	ALRRMCS2FRAME2 : ARRAY [1..3, 1..3] OF LREAL;
	ALRRFRAME22MCS : ARRAY [1..3, 1..3] OF LREAL;
	ALRRTCS2FRAME1 : ARRAY [1..3, 1..3] OF LREAL;
	ALRRTCS2FRAME2 : ARRAY [1..3, 1..3] OF LREAL;
	ALRRWCS2FRAME1 : ARRAY [1..3, 1..3] OF LREAL;
	ALRRWCS2FRAME2 : ARRAY [1..3, 1..3] OF LREAL;
	ALRRWCS2MCS : ARRAY [1..3, 1..3] OF LREAL;
	ALRRMCS2WCS : ARRAY [1..3, 1..3] OF LREAL;
	ALRXWCSFRAME1 : ARRAY [1..4] OF LREAL;
	ALRYWCSFRAME1 : ARRAY [1..4] OF LREAL;
	ALRZWCSFRAME1 : ARRAY [1..4] OF LREAL;
	ALRXWCSFRAME2 : ARRAY [1..4] OF LREAL;
	ALRYWCSFRAME2 : ARRAY [1..4] OF LREAL;
	ALRZWCSFRAME2 : ARRAY [1..4] OF LREAL;
	ALRXMCSFRAME1 : ARRAY [1..4] OF LREAL;
	ALRYMCSFRAME1 : ARRAY [1..4] OF LREAL;
	ALRZMCSFRAME1 : ARRAY [1..4] OF LREAL;
	ALRXMCSFRAME2 : ARRAY [1..4] OF LREAL;
	ALRYMCSFRAME2 : ARRAY [1..4] OF LREAL;
	ALRZMCSFRAME2 : ARRAY [1..4] OF LREAL;
	ALRXTCSFRAME1 : ARRAY [1..4] OF LREAL;
	ALRYTCSFRAME1 : ARRAY [1..4] OF LREAL;
	ALRZTCSFRAME1 : ARRAY [1..4] OF LREAL;
	ALRXTCSFRAME2 : ARRAY [1..4] OF LREAL;
	ALRYTCSFRAME2 : ARRAY [1..4] OF LREAL;
	ALRZTCSFRAME2 : ARRAY [1..4] OF LREAL;
	ALRPATH_MCS : ARRAY [1..100, 1..3] OF LREAL;
	ALRPATH_FRAME1 : ARRAY [1..100, 1..2] OF LREAL;
	ALRPATH_FRAME2 : ARRAY [1..100, 1..2] OF LREAL;
	XRESETPATHARRAY : BOOL := TRUE;
	ALRXTMP : ARRAY [1..3] OF LREAL;
	LRANGLEX : LREAL;
	LRANGLEY : LREAL;
	LRANGLEZ : LREAL;
	LRPROJLENGTHX : LREAL;
	LRPROJLENGTHY : LREAL;
	LRPROJLENGTHZ : LREAL;
	LRROTZ_FRAME1DEG : LREAL := 0;
	LRROTZ_FRAME1OLDDEG : LREAL := 0;
	LRROTZ_FRAME2DEG : LREAL := 0;
	LRROTZ_FRAME2OLDDEG : LREAL := 0;
	LRVALIDCOLOR : LREAL;
	ETRAFOERROR : L_IE1P_Error;
	XVALID : BOOL := FALSE;
	WSELECTFRAME1 : WORD;
	WSELECTFRAME2 : WORD;
	WSELECTFRAME1OLD : WORD;
	WSELECTFRAME2OLD : WORD;
	IFELD : INT := 1;
	USICOUNTERVAL : USINT := 0;
	AXSHOWPCS : ARRAY [1..16] OF BOOL;
	ALRPCSPOS_WCS : ARRAY [1..16, 1..6] OF LREAL;
	ALRRPCS2MCS : ARRAY [1..3, 1..3] OF LREAL;
	ALRRMCS2PCS : ARRAY [1..3, 1..3] OF LREAL;
	ALRRPCS2FRAME1 : ARRAY [1..3, 1..3] OF LREAL;
	ALRRPCS2FRAME2 : ARRAY [1..3, 1..3] OF LREAL;
	ALRXPCSFRAME1 : ARRAY [1..4] OF LREAL;
	ALRYPCSFRAME1 : ARRAY [1..4] OF LREAL;
	ALRZPCSFRAME1 : ARRAY [1..4] OF LREAL;
	ALRXPCSFRAME2 : ARRAY [1..4] OF LREAL;
	ALRYPCSFRAME2 : ARRAY [1..4] OF LREAL;
	ALRZPCSFRAME2 : ARRAY [1..4] OF LREAL;
	ALRMCS_T_WCS : ARRAY [1..4, 1..4] OF LREAL;
	ALRMCS_T_PCS : ARRAY [1..4, 1..4] OF LREAL;
	ALRWCS_T_PCS : ARRAY [1..4, 1..4] OF LREAL;
	XSHOWPCS : BOOL := FALSE;
	ESHOWPCS : L_MC4P_CoordSystem := L_MC4P_CoordSystem.PCS_1;
	XVISUHASPARAMETER : BOOL := FALSE;
	XSHOWMCS : BOOL := TRUE;
	XSHOWWCS : BOOL := FALSE;
	USIPATHCYCLES : USINT := 10;
	HEVENTCOMMCYCLE : Systypes.RTS_IEC_HANDLE := SysTypes.RTS_INVALID_HANDLE;
	HINTERFACECOMMCYCLE : Systypes.RTS_IEC_HANDLE := SysTypes.RTS_INVALID_HANDLE;
	ITFCALLBACK : CmpEventMgr.ICmpEventCallback;
	DWEVENTCOUNTER : DWORD;
	LRMCSPIXEL : LREAL := 50;
	LRTCSPIXEL : LREAL := 30;
	LRWCSPIXEL : LREAL := 50;
END_VAR
END_FUNCTION_BLOCK

METHOD COMMONINITIALIZE
END_METHOD

METHOD COMMONMAIN
END_METHOD

METHOD COORDSYSFRAME1
END_METHOD

METHOD COORDSYSFRAME2
END_METHOD

METHOD FB_EXIT : BOOL
VAR_INPUT
	BINCOPYCODE : BOOL;
END_VAR
END_METHOD

METHOD INITIALIZE
END_METHOD

METHOD KINEMATICFRAME1
END_METHOD

METHOD KINEMATICFRAME2
END_METHOD

METHOD PATH
END_METHOD

METHOD PATHFRAME1
END_METHOD

METHOD PATHFRAME2
END_METHOD

METHOD RECALCSCALINGS
END_METHOD

METHOD UPDATEORIENTATIONFRAME1
END_METHOD

METHOD UPDATEORIENTATIONFRAME2
END_METHOD

METHOD FB_INIT : BOOL
VAR_INPUT
	BINITRETAINS : BOOL;
	BINCOPYCODE : BOOL;
END_VAR
END_METHOD

METHOD EVENTCALLBACK : UDINT
VAR_INPUT
	PEVENTPARAM : POINTER TO EventParam;
END_VAR
END_METHOD

METHOD REGISTEREVENT
END_METHOD

METHOD UNREGISTEREVENT
END_METHOD

(* ---- L_MC4P_WRITEBOOLPARAMETER.pou ---- *)
FUNCTION_BLOCK L_MC4P_WRITEBOOLPARAMETER EXTENDS L_MC4P_Template_AG_KIN
VAR_INPUT
	XEXECUTE : BOOL;
	DIPARAMETERNUMBER : DINT;
	XVALUE : BOOL;
END_VAR
VAR_OUTPUT
	XDONE : BOOL;
	XBUSY : BOOL;
	XERROR : BOOL;
	EERRORID : L_IE1P_Error;
END_VAR
VAR
	XEXECUTEOLD : BOOL := FALSE;
	XRESETOUTPUT : BOOL := FALSE;
	WERRORID_INT : WORD;
END_VAR
END_FUNCTION_BLOCK

METHOD FB_RESET : BOOL
END_METHOD

(* ---- L_MC4P_WRITEPARAMETER.pou ---- *)
FUNCTION_BLOCK L_MC4P_WRITEPARAMETER EXTENDS L_MC4P_Template_AG_KIN
VAR_INPUT
	XEXECUTE : BOOL;
	DIPARAMETERNUMBER : DINT;
	LRVALUE : LREAL;
END_VAR
VAR_OUTPUT
	XDONE : BOOL;
	XBUSY : BOOL;
	XERROR : BOOL;
	EERRORID : L_IE1P_Error;
END_VAR
VAR
	XEXECUTEOLD : BOOL := FALSE;
	XRESETOUTPUT : BOOL := FALSE;
	WERRORID_INT : WORD;
END_VAR
END_FUNCTION_BLOCK

METHOD FB_RESET : BOOL
END_METHOD

(* ---- L_MC4P_WRITEPATHFILE_INTERNAL.pou ---- *)
FUNCTION_BLOCK L_MC4P_WRITEPATHFILE_INTERNAL
VAR_INPUT
	XEXECUTE : BOOL;
	SFILENAME : STRING;
	SFILEADRES : STRING := '\USBStorage\IPC\PLC\MovePathData\';
	DINUMOFLINES : DINT := 200;
END_VAR
VAR_OUTPUT
	XDONE : BOOL;
	XBUSY : BOOL;
	XCOMMANDABORTED : BOOL;
	XERROR : BOOL;
	EERRORID : L_IE1P_Error;
END_VAR
VAR_IN_OUT
	ASPATHFILE : ARRAY [1..200] OF STRING(255);
END_VAR
VAR
	WSTATE : WORD;
	XNEWFILE_INT : BOOL;
	DILINENO_INT : DINT;
	DINUMOFLINES_INT : DINT;
	UDIPOSINFILE : UDINT;
	FB_SEMA : L_MC1P_CriticalSection;
	REQUESTSINFO : DWORD;
	REQUESTSINFO_OLD : DWORD;
	DWRTRIG : DWORD;
	DWFTRIG : DWORD;
	SFILE_INT : STRING := '';
	WTASKCYCLECOUNTER : WORD := 0;
	XLOWTASKBUSY_INT : BOOL;
	XLOWTASKDONE_INT : BOOL;
	XLOWTASKERROR_INT : BOOL;
	ELOWTASKERRORID_INT : L_IE1P_Error;
	RES : SYSFILE.RTS_IEC_ResULT;
	HFILE : SYSFILE.RTS_IEC_HANDLE;
	UDILENGTHFILE : UDINT;
	UDIFSIZE : UDINT;
	XTESTINMOTIONTASK : BOOL := FALSE;
	ILINELEN_INT : INT;
	XERROR_TIMEOUT : BOOL;
	FILDCR : FILE.DirCreate;
	SLINE : STRING(255);
	XDECODEINMOTIONTASK : BOOL;
END_VAR
END_FUNCTION_BLOCK

METHOD ABORTFB : UDINT
END_METHOD

METHOD CALL_ERRORHANDLER
END_METHOD

METHOD CALL_FBMETHODS
END_METHOD

METHOD CALL_OUTPUT
END_METHOD

METHOD CALL_REQUESTS_EXT
END_METHOD

METHOD CALL_RESETCOMMANDS
END_METHOD

METHOD CALL_RESETOUTPUT
END_METHOD

METHOD CALL_STATEMACHINE
END_METHOD

METHOD RESETREADDATA
END_METHOD

METHOD CALL_WRITEFILE
END_METHOD

METHOD EXECUTEFREERUNTASK
END_METHOD

METHOD MAIN
END_METHOD

METHOD ABORT : UDINT
END_METHOD

METHOD EXECUTE : UDINT
END_METHOD

(* ---- MC_ADDAXISTOGROUP.pou ---- *)
FUNCTION_BLOCK MC_ADDAXISTOGROUP EXTENDS L_MC4P_Template_AG_KIN
VAR_INPUT
	EXECUTE : BOOL;
	IDENTINGROUP : IDENT_IN_GROUP_REF;
END_VAR
VAR_OUTPUT
	DONE : BOOL;
	BUSY : BOOL;
	ERROR : BOOL;
	ERRORID : L_IE1P_Error;
END_VAR
VAR_IN_OUT
	AXIS : AXIS_REF;
END_VAR
VAR
	XERRORINTERN : BOOL;
	EERRORIDINTERN : L_IE1P_Error := L_IE1P_Error.NoError;
	XEXECUTEOLD : BOOL;
	XRESETOUTPUT : BOOL;
	PSDUMMY : POINTER TO STRING;
	PAXIS : POINTER TO POINTER TO AXIS_REF;
END_VAR
END_FUNCTION_BLOCK

(* ---- MC_GROUPDISABLE.pou ---- *)
FUNCTION_BLOCK MC_GROUPDISABLE EXTENDS L_MC4P_Template_AG_REF
VAR_INPUT
	EXECUTE : BOOL;
END_VAR
VAR_OUTPUT
	DONE : BOOL;
	BUSY : BOOL;
	ERROR : BOOL;
	ERRORID : L_IE1P_Error;
END_VAR
VAR
	XEXECUTEOLD : BOOL;
	IDX : WORD;
	XRESETOUTPUT : BOOL;
	XVIRTAXISENABLED : BOOL;
	PXDUMMY : POINTER TO BOOL;
	PAXESGROUP : POINTER TO AXES_GROUP_KIN;
	WDISABLECNTR : WORD;
	WDISABLECNTRMAX : WORD := 50;
	XREADYFORDISABLE : BOOL;
	WSTATE : WORD;
	XDOWHILE : BOOL;
	ICNT : INT;
END_VAR
END_FUNCTION_BLOCK

(* ---- MC_GROUPENABLE.pou ---- *)
FUNCTION_BLOCK MC_GROUPENABLE EXTENDS L_MC4P_Template_AG_REF
VAR_INPUT
	EXECUTE : BOOL;
END_VAR
VAR_OUTPUT
	DONE : BOOL;
	BUSY : BOOL;
	ERROR : BOOL;
	ERRORID : L_IE1P_Error;
END_VAR
VAR
	XEXECUTEOLD : BOOL;
	IDX : WORD;
	XRESETOUTPUT : BOOL;
	XREALAXISENABLED : BOOL;
	XREALAXISSTANDSTILL : BOOL;
	XVIRTAXISENABLED : BOOL;
	WSTEP : WORD;
	PXDUMMY : POINTER TO BOOL;
	ALRKARTPOS : ARRAY [1..6] OF LREAL;
	ALRACTAXESPOS : ARRAY [1..6] OF LREAL;
	ALRCALCULATEDAXESPOS : ARRAY [1..6] OF LREAL;
	ALRAXESPOSDIFF : ARRAY [1..6] OF LREAL;
	PAXESGROUP : POINTER TO AXES_GROUP_KIN;
	XERRORINTERN : BOOL;
	EERRORIDINTERN : L_IE1P_Error;
	EERRORIDINTERN2 : L_IE1P_Error;
	SCERROR : L_MC4P_ErrorStruct;
	SCINFO : L_MC4P_TrafoInfo;
END_VAR
END_FUNCTION_BLOCK

METHOD FB_INIT : BOOL
VAR_INPUT
	BINITRETAINS : BOOL;
	BINCOPYCODE : BOOL;
END_VAR
END_METHOD

(* ---- MC_GROUPHOME.pou ---- *)
FUNCTION_BLOCK MC_GROUPHOME EXTENDS L_MC4P_Template_AG_KIN_Licence
VAR_INPUT
	EXECUTE : BOOL;
	POSITION : ARRAY [1..12] OF LREAL;
	HOMINGORDER : ARRAY [1..12] OF L_MC4P_HomingOrder := [12(0)];
	HOMEABSSWITCH : ARRAY [1..12] OF BOOL;
	USEEXTPARAMETER : ARRAY [1..12] OF BOOL;
	EXTPARAMETER : ARRAY [1..12] OF L_MC1P_HomeParameter;
	EXTTP : ARRAY [1..12] OF MC_TRIGGER_REF;
END_VAR
VAR_OUTPUT
	DONE : BOOL;
	BUSY : BOOL;
	ACTIVE : BOOL;
	COMMANDABORTED : BOOL;
	ERROR : BOOL;
	ERRORID : L_IE1P_Error;
	AXISDONE : ARRAY [1..12] OF BOOL;
END_VAR
VAR
	HOME : L_MC4P_GroupHome_Internal;
END_VAR
END_FUNCTION_BLOCK

(* ---- MC_GROUPREADACTUALACCELERATION.pou ---- *)
FUNCTION_BLOCK MC_GROUPREADACTUALACCELERATION EXTENDS L_MC4P_Template_AG_KIN
VAR_INPUT
	ENABLE : BOOL;
	COORDSYSTEM : L_MC4P_CoordSystem;
END_VAR
VAR_OUTPUT
	VALID : BOOL;
	BUSY : BOOL;
	ERROR : BOOL;
	ERRORID : L_IE1P_Error;
	ACCELERATION : ARRAY [1..12] OF LREAL;
	PATHACCELERATION : LREAL;
END_VAR
VAR
	IDX : WORD;
	XENABLEOLD : BOOL;
	PCOORDTRAFO : POINTER TO L_MC4P_CoordTrafo;
	ALRACCELERATIONTMP1 : ARRAY [1..6] OF LREAL;
	ALRACCELERATIONTMP2 : ARRAY [1..6] OF LREAL;
	ALRVELOCITYTMP1 : ARRAY [1..6] OF LREAL;
	ALRVELOCITYTMP2 : ARRAY [1..6] OF LREAL;
	ALRPOSITIONTMP : ARRAY [1..6] OF LREAL;
	ALRPOSVEKPCS2TCS : ARRAY [1..3] OF LREAL;
	ROT_MAT : ARRAY [1..3, 1..3] OF LREAL;
	ROT_MATT : ARRAY [1..3, 1..3] OF LREAL;
	ALRTMP : ARRAY [1..3] OF LREAL;
	T1 : LREAL;
	T5 : LREAL;
	T6 : LREAL;
	T7 : LREAL;
	T13 : LREAL;
	T20 : LREAL;
	T21 : LREAL;
	T26 : LREAL;
	X : LREAL;
	Y : LREAL;
	XPUNKT : LREAL;
	YPUNKT : LREAL;
	XPUNKTPUNKT : LREAL;
	YPUNKTPUNKT : LREAL;
END_VAR
END_FUNCTION_BLOCK

(* ---- MC_GROUPREADACTUALPOSITION.pou ---- *)
FUNCTION_BLOCK MC_GROUPREADACTUALPOSITION EXTENDS L_MC4P_Template_AG_KIN
VAR_INPUT
	ENABLE : BOOL;
	COORDSYSTEM : L_MC4P_CoordSystem;
END_VAR
VAR_OUTPUT
	VALID : BOOL;
	BUSY : BOOL;
	ERROR : BOOL;
	ERRORID : L_IE1P_Error;
	POSITION : ARRAY [1..12] OF LREAL;
END_VAR
VAR
	XUSESETVALUES : BOOL := FALSE;
	READPOSITION : L_MC4P_GroupReadActualPosition_Internal;
	USESETVALUES : BOOL;
END_VAR
END_FUNCTION_BLOCK

(* ---- MC_GROUPREADACTUALVELOCITY.pou ---- *)
FUNCTION_BLOCK MC_GROUPREADACTUALVELOCITY EXTENDS L_MC4P_Template_AG_KIN
VAR_INPUT
	ENABLE : BOOL;
	COORDSYSTEM : L_MC4P_CoordSystem;
END_VAR
VAR_OUTPUT
	VALID : BOOL;
	BUSY : BOOL;
	ERROR : BOOL;
	ERRORID : L_IE1P_Error;
	VELOCITY : ARRAY [1..12] OF LREAL;
	PATHVELOCITY : LREAL;
END_VAR
VAR
	XUSESETVALUES : BOOL := FALSE;
	READVEL : L_MC4P_GroupReadActualVelocity_Internal;
	USESETVALUES : BOOL;
END_VAR
END_FUNCTION_BLOCK

(* ---- MC_GROUPREADERROR.pou ---- *)
FUNCTION_BLOCK MC_GROUPREADERROR EXTENDS L_MC4P_Template_AG_REF
VAR_INPUT
	ENABLE : BOOL;
END_VAR
VAR_OUTPUT
	VALID : BOOL;
	BUSY : BOOL;
	ERROR : BOOL;
	ERRORID : L_IE1P_Error;
	GROUPWARNING : BOOL;
	GROUPERROR : BOOL;
	GROUPERRORID : L_IE1P_Error;
	PINSTANCENAME : POINTER TO STRING := ADR(NoError);
	TIMESTAMP : TIME;
END_VAR
VAR
	XENABLEOLD : BOOL;
	NOERROR : STRING := '';
END_VAR
END_FUNCTION_BLOCK

(* ---- MC_GROUPREADSTATUS.pou ---- *)
FUNCTION_BLOCK MC_GROUPREADSTATUS EXTENDS L_MC4P_Template_AG_KIN
VAR_INPUT
	ENABLE : BOOL;
END_VAR
VAR_OUTPUT
	VALID : BOOL;
	BUSY : BOOL;
	ERROR : BOOL;
	ERRORID : L_IE1P_Error;
	GROUPMOVING : BOOL;
	GROUPHOMING : BOOL;
	GROUPERRORSTOP : BOOL;
	GROUPSTANDBY : BOOL;
	GROUPSTOPPING : BOOL;
	GROUPDISABLED : BOOL;
	CONSTANTVELOCITY : BOOL;
	ACCELERATING : BOOL;
	DECELERATING : BOOL;
	INPOSITION : BOOL;
	STANDSTILL : BOOL;
END_VAR
VAR
	READSTATUS : L_MC4P_GroupReadStatus_Internal;
END_VAR
END_FUNCTION_BLOCK

(* ---- MC_GROUPRESET.pou ---- *)
FUNCTION_BLOCK MC_GROUPRESET EXTENDS L_MC4P_Template_AG_REF
VAR_INPUT
	EXECUTE : BOOL;
END_VAR
VAR_OUTPUT
	DONE : BOOL;
	BUSY : BOOL;
	ERROR : BOOL;
	ERRORID : L_IE1P_Error;
END_VAR
VAR
	GROUPRESET : L_MC4P_GroupReset_Internal;
END_VAR
END_FUNCTION_BLOCK

(* ---- MC_GROUPSETPOSITION.pou ---- *)
FUNCTION_BLOCK MC_GROUPSETPOSITION EXTENDS L_MC4P_Template_AG_KIN
VAR_INPUT
	EXECUTE : BOOL;
	POSITION : ARRAY [1..12] OF LREAL;
	RELATIVE : BOOL := FALSE;
END_VAR
VAR_OUTPUT
	DONE : BOOL;
	BUSY : BOOL;
	ACTIVE : BOOL;
	ERROR : BOOL;
	ERRORID : L_IE1P_Error;
END_VAR
VAR
	SETPOSITION : L_MC4P_GroupSetPosition_Internal;
END_VAR
END_FUNCTION_BLOCK

(* ---- MC_GROUPSTOP.pou ---- *)
FUNCTION_BLOCK MC_GROUPSTOP EXTENDS L_MC4P_Template_AG_KIN_Licence
VAR_INPUT
	EXECUTE : BOOL;
	DECELERATION : LREAL;
	JERK : LREAL;
END_VAR
VAR_OUTPUT
	DONE : BOOL;
	BUSY : BOOL;
	ACTIVE : BOOL;
	COMMANDABORTED : BOOL;
	ERROR : BOOL;
	ERRORID : L_IE1P_Error;
END_VAR
VAR
	STOP : L_MC4P_GroupStop_Internal;
END_VAR
END_FUNCTION_BLOCK

(* ---- MC_MOVECIRCULARABSOLUTE.pou ---- *)
FUNCTION_BLOCK MC_MOVECIRCULARABSOLUTE EXTENDS L_MC4P_Template_MoveLicence
VAR_INPUT
	EXECUTE : BOOL;
	CIRCMODE : L_MC4P_CircMode;
	AUXPOINT : ARRAY [1..12] OF LREAL;
	ENDPOINT : ARRAY [1..12] OF LREAL;
	PATHCHOICE : MC_CIRC_PATHCHOICE;
	VELOCITY : LREAL;
	ACCELERATION : LREAL;
	DECELERATION : LREAL;
	JERK : LREAL;
	COORDSYSTEM : L_MC4P_CoordSystem;
	BUFFERMODE : MC_BUFFER_MODE;
	TRANSITIONMODE : MC_TRANSITION_MODE;
	TRANSITIONPARAMETER : ARRAY [1..12] OF LREAL := [12(0)];
	AEAUXMODE : ARRAY [1..6] OF L_MC4P_AuxMode;
	ORIENTATIONMODE : L_MC4P_Orientation_Mode := L_MC4P_Orientation_Mode.ShortestSpacialWay;
	DIRECTION : ARRAY [4..6] OF MC_DIRECTION := [3(MC_DIRECTION.mcShortestWay)];
END_VAR
VAR_OUTPUT
	DONE : BOOL;
	BUSY : BOOL;
	ACTIVE : BOOL;
	COMMANDABORTED : BOOL;
	ERROR : BOOL;
	ERRORID : L_IE1P_Error;
END_VAR
VAR
	MOVECIRC : L_MC4P_MoveCircularAbsolute_Internal;
	PMOVE : POINTER TO L_MC4P_MoveContPath;
END_VAR
END_FUNCTION_BLOCK

(* ---- MC_MOVECIRCULARRELATIVE.pou ---- *)
FUNCTION_BLOCK MC_MOVECIRCULARRELATIVE EXTENDS L_MC4P_Template_MoveLicence
VAR_INPUT
	EXECUTE : BOOL;
	CIRCMODE : L_MC4P_CircMode;
	AUXPOINT : ARRAY [1..12] OF LREAL;
	ENDPOINT : ARRAY [1..12] OF LREAL;
	PATHCHOICE : MC_CIRC_PATHCHOICE;
	VELOCITY : LREAL;
	ACCELERATION : LREAL;
	DECELERATION : LREAL;
	JERK : LREAL;
	COORDSYSTEM : L_MC4P_CoordSystem;
	BUFFERMODE : MC_BUFFER_MODE;
	TRANSITIONMODE : MC_TRANSITION_MODE;
	TRANSITIONPARAMETER : ARRAY [1..12] OF LREAL := [12(0)];
	AEAUXMODE : ARRAY [1..6] OF L_MC4P_AuxMode;
	ORIENTATIONMODE : L_MC4P_Orientation_Mode := L_MC4P_Orientation_Mode.ShortestSpacialWay;
	DIRECTION : ARRAY [4..6] OF MC_DIRECTION := [3(MC_DIRECTION.mcShortestWay)];
END_VAR
VAR_OUTPUT
	DONE : BOOL;
	BUSY : BOOL;
	ACTIVE : BOOL;
	COMMANDABORTED : BOOL;
	ERROR : BOOL;
	ERRORID : L_IE1P_Error;
END_VAR
VAR
	MOVECIRC : L_MC4P_MoveCircularRelative_Internal;
	PMOVE : POINTER TO L_MC4P_MoveContPath;
END_VAR
END_FUNCTION_BLOCK

(* ---- MC_MOVEDIRECTABSOLUTE.pou ---- *)
FUNCTION_BLOCK MC_MOVEDIRECTABSOLUTE EXTENDS L_MC4P_Template_MoveLicence
VAR_INPUT
	EXECUTE : BOOL;
	POSITION : ARRAY [1..12] OF LREAL;
	COORDSYSTEM : L_MC4P_CoordSystem;
	BUFFERMODE : MC_BUFFER_MODE;
	TRANSITIONMODE : MC_TRANSITION_MODE;
	TRANSITIONPARAMETER : ARRAY [1..12] OF LREAL := [12(0)];
	AITARGETCONFIGURATION : ARRAY [1..6] OF INT;
	DIRECTION : ARRAY [1..6] OF MC_DIRECTION := [6(MC_DIRECTION.mcShortestWay)];
END_VAR
VAR_OUTPUT
	DONE : BOOL;
	BUSY : BOOL;
	ACTIVE : BOOL;
	COMMANDABORTED : BOOL;
	ERROR : BOOL;
	ERRORID : L_IE1P_Error;
END_VAR
VAR
	MOVEDIRECT : L_MC4P_MoveDirectAbsolute_Internal;
	PMOVE : POINTER TO L_MC4P_MoveContPath;
END_VAR
END_FUNCTION_BLOCK

(* ---- MC_MOVEDIRECTRELATIVE.pou ---- *)
FUNCTION_BLOCK MC_MOVEDIRECTRELATIVE EXTENDS L_MC4P_Template_MoveLicence
VAR_INPUT
	EXECUTE : BOOL;
	DISTANCE : ARRAY [1..12] OF LREAL;
	COORDSYSTEM : L_MC4P_CoordSystem;
	BUFFERMODE : MC_BUFFER_MODE;
	TRANSITIONMODE : MC_TRANSITION_MODE;
	TRANSITIONPARAMETER : ARRAY [1..12] OF LREAL := [12(0)];
	AITARGETCONFIGURATION : ARRAY [1..6] OF INT;
	DIRECTION : ARRAY [1..6] OF MC_DIRECTION := [6(MC_DIRECTION.mcShortestWay)];
END_VAR
VAR_OUTPUT
	DONE : BOOL;
	BUSY : BOOL;
	ACTIVE : BOOL;
	COMMANDABORTED : BOOL;
	ERROR : BOOL;
	ERRORID : L_IE1P_Error;
END_VAR
VAR
	MOVEDIRECT : L_MC4P_MoveDirectRelative_Internal;
	PMOVE : POINTER TO L_MC4P_MoveContPath;
END_VAR
END_FUNCTION_BLOCK

(* ---- MC_MOVELINEARABSOLUTE.pou ---- *)
FUNCTION_BLOCK MC_MOVELINEARABSOLUTE EXTENDS L_MC4P_Template_MoveLicence
VAR_INPUT
	EXECUTE : BOOL;
	POSITION : ARRAY [1..12] OF LREAL;
	VELOCITY : LREAL;
	ACCELERATION : LREAL;
	DECELERATION : LREAL;
	JERK : LREAL;
	COORDSYSTEM : L_MC4P_CoordSystem;
	BUFFERMODE : MC_BUFFER_MODE;
	TRANSITIONMODE : MC_TRANSITION_MODE;
	TRANSITIONPARAMETER : ARRAY [1..12] OF LREAL := [12(0)];
	AEAUXMODE : ARRAY [1..6] OF L_MC4P_AuxMode;
	ORIENTATIONMODE : L_MC4P_Orientation_Mode := L_MC4P_Orientation_Mode.ShortestSpacialWay;
	DIRECTION : ARRAY [4..6] OF MC_DIRECTION := [3(MC_DIRECTION.mcShortestWay)];
END_VAR
VAR_OUTPUT
	DONE : BOOL;
	BUSY : BOOL;
	ACTIVE : BOOL;
	COMMANDABORTED : BOOL;
	ERROR : BOOL;
	ERRORID : L_IE1P_Error;
END_VAR
VAR
	MOVELIN : L_MC4P_MoveLinearAbsolute_Internal;
	PMOVE : POINTER TO L_MC4P_MoveContPath;
END_VAR
END_FUNCTION_BLOCK

(* ---- MC_MOVELINEARRELATIVE.pou ---- *)
FUNCTION_BLOCK MC_MOVELINEARRELATIVE EXTENDS L_MC4P_Template_MoveLicence
VAR_INPUT
	EXECUTE : BOOL;
	DISTANCE : ARRAY [1..12] OF LREAL;
	VELOCITY : LREAL;
	ACCELERATION : LREAL;
	DECELERATION : LREAL;
	JERK : LREAL;
	COORDSYSTEM : L_MC4P_CoordSystem;
	BUFFERMODE : MC_BUFFER_MODE;
	TRANSITIONMODE : MC_TRANSITION_MODE;
	TRANSITIONPARAMETER : ARRAY [1..12] OF LREAL := [12(0)];
	AEAUXMODE : ARRAY [1..6] OF L_MC4P_AuxMode;
	ORIENTATIONMODE : L_MC4P_Orientation_Mode := L_MC4P_Orientation_Mode.ShortestSpacialWay;
	DIRECTION : ARRAY [4..6] OF MC_DIRECTION := [3(MC_DIRECTION.mcShortestWay)];
END_VAR
VAR_OUTPUT
	DONE : BOOL;
	BUSY : BOOL;
	ACTIVE : BOOL;
	COMMANDABORTED : BOOL;
	ERROR : BOOL;
	ERRORID : L_IE1P_Error;
END_VAR
VAR
	MOVELIN : L_MC4P_MoveLinearRelative_Internal;
	PMOVE : POINTER TO L_MC4P_MoveContPath;
END_VAR
END_FUNCTION_BLOCK

(* ---- MC_MOVEPATH.pou ---- *)
FUNCTION_BLOCK MC_MOVEPATH EXTENDS L_MC4P_Template_AG_KIN_Licence
VAR_INPUT
	PATHREF : MC_PATH_REF;
	EXECUTE : BOOL;
	VELOCITY : LREAL;
	ACCELERATION : LREAL;
	DECELERATION : LREAL;
	JERK : LREAL;
	COORDSYSTEM : L_MC4P_CoordSystem;
	BUFFERMODE : MC_BUFFER_MODE;
	TRANSITIONMODE : MC_TRANSITION_MODE;
	TRANSITIONPARAMETER : ARRAY [1..12] OF LREAL := [12(0)];
	MODE : WORD;
	ACKPATHHALT : BOOL;
	MACKNOWLEDGE : BOOL;
	ACKBLOCKSEARCH : BOOL;
END_VAR
VAR_OUTPUT
	DONE : BOOL;
	BUSY : BOOL;
	ACTIVE : BOOL;
	COMMANDABORTED : BOOL;
	ERROR : BOOL;
	ERRORID : L_IE1P_Error;
	SOURCELINENO : LINT;
	SOURCELINE : STRING;
	MFUNCTION : WORD;
	WAITINGFORMACKNOWLEDGE : BOOL;
	NEWVALUEMFUNCTION : BOOL;
	WAITINGFORACKPATHHALT : BOOL;
	WAITINGFORACKBLOCKSEARCH : BOOL;
END_VAR
VAR
	LRVELOCITY_INT : LREAL;
	LRACCELERATION_INT : LREAL;
	LRDECELERATION_INT : LREAL;
	LRJERK_INT : LREAL;
	ECOORDSYSTEM_INT : L_MC4P_CoordSystem;
	EBUFFERMODE_INT : MC_BUFFER_MODE;
	ETRANSITIONMODE_INT : MC_TRANSITION_MODE;
	ALRTRANSITIONPARAMETER_INT : ARRAY [1..12] OF LREAL := [12(0)];
	EMODE_INT : WORD;
	DIACKPATHHALT_INT : DINT;
	XERROR_OLD : BOOL;
	XPATHREFVALID : BOOL;
	XWPATHREFID : __XWORD;
	DWPATHREFSTATUS : DWORD;
	XPATHREFERROR : BOOL;
	XPATHREFDONE : BOOL;
	XPATHREFBUSY : BOOL;
	XPATHREFCOMMANDABORTED : BOOL;
	XPATHREFDECODING : BOOL;
	XPATHREFINTERPRETERHALT : BOOL;
	XINTERPRETERHALTACKED : BOOL;
	XPATHREFINTERPRETERHALTAPPL : BOOL;
	XPATHREFDATAACTIVE : BOOL;
	APELEMENT : ARRAY [1..GVL_MovePath.gciNumOfDecodeAsciiData] OF POINTER TO L_MC4P_Parameter_MCMove;
	PELEMENT : POINTER TO L_MC4P_Parameter_MCMove;
	SCINITELEMENT : L_MC4P_Parameter_MCMove;
	IPATHSTARTNO : INT;
	IPATHDATASIZE : UDINT;
	LIFILELINENO : LINT;
	XUPDATESOURCE : BOOL;
	XBUSY_INT : BOOL;
	XDONE_INT : BOOL;
	XCOMMANDABORTED_INT : BOOL;
	XWAITFORDONE : BOOL;
	XERROR_INT : BOOL;
	REQUESTSINFO : DWORD;
	REQUESTSINFO_OLD : DWORD;
	DWRTRIG : DWORD;
	DWFTRIG : DWORD;
	XRESETOUTPUTS : BOOL;
	XSEGMENTACTIVE_OLD : BOOL;
	MFUNCTION_OLD : WORD;
	XMACKNOWLEDGEACTIVE : BOOL;
	XSETFIRSTSOURCELINE_LOCK : BOOL;
	XWPATHREFID_LOCK : __XWORD;
	XSETPATHDATAACTIVE_LOCK : BOOL;
	XUNLOCKPATHREF : BOOL;
	DWSTATE_INT : DWORD;
	IEXECUTEELEMENTSIZE : INT;
	IEXECUTEELEMENTSIZE_LOCK : INT;
	XERRORINVALIDPATHREF : BOOL;
	XERRORPATHREFINUSE : BOOL;
	XMOVECONTPATHDONE : BOOL;
	XMOVECONTPATHBUSY : BOOL;
	XMOVECONTPATHWAITFORINTERPRETER : BOOL;
	XMOVECONTPATHCOMMANDABORTED : BOOL;
	XMOVECONTPATHCOMMANDABORTEDATHALT : BOOL;
	XMOVECONTPATHERROR : BOOL;
	EMOVECONTPATHERRORID : L_IE1P_Error;
	IACKNMOVECONTPATHNO : INT;
	FB_MOVECONTPATHCONTROL : L_MC1P_StackControlArray := STRUCT(iMaxLegth := L_MC4P_Constants.ciNumOfMoveContPath);
	XMOVECONTPATHACTIVELOCK : BOOL;
	XDISABLEMOVECONTPATH : BOOL;
	REFFBSTORE : REFERENCE TO L_MC4P_MovePathStore;
	XOPTIMISEDPATHPREPARATION_INT : BOOL := TRUE;
	IELEMENTSIZECHECKFORPROFILECALC : INT;
	INUMOFGROUPSFORCALCPROFILE : INT;
	INUMOFSEGMENTINGROUPFORCALCPROFILE : INT;
	LRTIMEGROUPFORCALCPROFILE_OLD : LREAL;
	LRTIMEGROUPFORCALCPROFILE : LREAL;
	IMAXNUMOFSEGMENTINGROUPFORCALCPROFILE : INT := 7;
	LRMAXTIMEGROUPFORCALCPROFILE : LREAL := 0.7;
	XMOTIONREQUESTED : BOOL;
	XBLOCKSEARCHACKACTIVE : BOOL;
	XBLOCKFOUND : BOOL;
	_XSEMALOCKED : BOOL;
	FBREADPOS : MC_GroupReadActualPosition;
	XOPTIMISEDPATHPREPARATION : BOOL;
END_VAR
END_FUNCTION_BLOCK

METHOD CALL_ALLOCPOINTADR
END_METHOD

METHOD CALL_DISABLEMOVECONTPATH
VAR_IN_OUT
	AXESGROUP : AXES_GROUP_KIN;
END_VAR
END_METHOD

METHOD CALL_ERRORHANDLER
VAR_IN_OUT
	AXESGROUP : AXES_GROUP_KIN;
END_VAR
END_METHOD

METHOD CALL_FBMETHODS
VAR_IN_OUT
	AXESGROUP : AXES_GROUP_KIN;
END_VAR
END_METHOD

METHOD CALL_FB_MOVECONTPATH
VAR_IN_OUT
	AXESGROUP : AXES_GROUP_KIN;
END_VAR
END_METHOD

METHOD CALL_OUTPUT
END_METHOD

METHOD CALL_REQUESTS_EXT
END_METHOD

METHOD CALL_RESETCOMMANDS
END_METHOD

METHOD CALL_RESETOUTPUT
END_METHOD

METHOD CALL_STATEMACHINE
VAR_IN_OUT
	AXESGROUP : AXES_GROUP_KIN;
END_VAR
END_METHOD

METHOD CALL_UNLOCKPATHDATA
VAR_IN_OUT
	AXESGROUP : AXES_GROUP_KIN;
END_VAR
END_METHOD

METHOD FUN_ACKNLASTELEMENT : BOOL
VAR_INPUT
	PELEMENT : POINTER TO L_MC4P_Parameter_MCMove;
	IDX : INT;
END_VAR
END_METHOD

METHOD FUN_ACKNOWLEDGEELEMENT
VAR_INPUT
	IELEMENTNO : INT := 1;
END_VAR
END_METHOD

METHOD FUN_INITELEMENT
VAR_IN_OUT
	AXESGROUP : AXES_GROUP_KIN;
	SCPARELEMENT : L_MC4P_Parameter_MCMove;
END_VAR
END_METHOD

METHOD FUN_SEARCHFINALELEMENT : BOOL
END_METHOD

METHOD FB_INIT : BOOL
VAR_INPUT
	BINITRETAINS : BOOL;
	BINCOPYCODE : BOOL;
END_VAR
END_METHOD

METHOD CALL_PATHREFINFO
END_METHOD

METHOD CALL_INIT
END_METHOD

METHOD CALL_S000_CYCLIC
VAR_IN_OUT
	AXESGROUP : AXES_GROUP_KIN;
END_VAR
END_METHOD

(* ---- MC_READCARTESIANTRANSFORM.pou ---- *)
FUNCTION_BLOCK MC_READCARTESIANTRANSFORM EXTENDS L_MC4P_Template_AG_KIN
VAR_INPUT
	ENABLE : BOOL;
	COORDSYSTEM : L_MC4P_CoordSystem;
END_VAR
VAR_OUTPUT
	VALID : BOOL;
	BUSY : BOOL;
	ERROR : BOOL;
	ERRORID : L_IE1P_Error;
	TRANSX : LREAL;
	TRANSY : LREAL;
	TRANSZ : LREAL;
	ROTANGLE1 : LREAL;
	ROTANGLE2 : LREAL;
	ROTANGLE3 : LREAL;
END_VAR
VAR
	PCOORDTRAFO : POINTER TO L_MC4P_CoordTrafo;
	XENABLEOLD : BOOL;
END_VAR
END_FUNCTION_BLOCK

(* ---- MC_READCOORDINATETRANSFORM.pou ---- *)
FUNCTION_BLOCK MC_READCOORDINATETRANSFORM EXTENDS L_MC4P_Template_AG_KIN
VAR_INPUT
	ENABLE : BOOL;
	COORDSYSTEM : L_MC4P_CoordSystem;
END_VAR
VAR_OUTPUT
	VALID : BOOL;
	BUSY : BOOL;
	ERROR : BOOL;
	ERRORID : L_IE1P_Error;
	COORDTRANSFORM : MC_COORD_REF;
END_VAR
VAR
	PCOORDTRAFO : POINTER TO L_MC4P_CoordTrafo;
	XENABLEOLD : BOOL;
END_VAR
END_FUNCTION_BLOCK

(* ---- MC_REMOVEAXISFROMGROUP.pou ---- *)
FUNCTION_BLOCK MC_REMOVEAXISFROMGROUP EXTENDS L_MC4P_Template_AG_KIN
VAR_INPUT
	EXECUTE : BOOL;
	IDENTINGROUP : IDENT_IN_GROUP_REF;
END_VAR
VAR_OUTPUT
	DONE : BOOL;
	BUSY : BOOL;
	ERROR : BOOL;
	ERRORID : L_IE1P_Error;
END_VAR
VAR
	XERRORINTERN : BOOL;
	EERRORIDINTERN : L_IE1P_Error := L_IE1P_Error.NoError;
	XEXECUTEOLD : BOOL;
	XRESETOUTPUT : BOOL;
	PSDUMMY : POINTER TO STRING;
	DWINTERNALERRORID : DWORD;
END_VAR
END_FUNCTION_BLOCK

(* ---- MC_SETCARTESIANTRANSFORM.pou ---- *)
FUNCTION_BLOCK MC_SETCARTESIANTRANSFORM EXTENDS L_MC4P_Template_AG_KIN
VAR_INPUT
	EXECUTE : BOOL;
	COORDSYSTEM : L_MC4P_CoordSystem;
	TRANSX : LREAL;
	TRANSY : LREAL;
	TRANSZ : LREAL;
	ROTANGLE1 : LREAL;
	ROTANGLE2 : LREAL;
	ROTANGLE3 : LREAL;
END_VAR
VAR_OUTPUT
	DONE : BOOL;
	BUSY : BOOL;
	ACTIVE : BOOL;
	COMMANDABORTED : BOOL;
	ERROR : BOOL;
	ERRORID : L_IE1P_Error;
END_VAR
VAR
	PCOORDTRAFO : POINTER TO L_MC4P_CoordTrafo;
	XEXECUTEOLD : BOOL;
	XRESETOUTPUT : BOOL;
	ISTATE : INT;
	BSTATEMACHINE : BOOL;
	PTRACKINGPARAM : POINTER TO L_MC4P_PCSTrackParam;
	ALRPARAMFREEZE : ARRAY [1..6] OF LREAL;
	AXPARACCESSIBLE : ARRAY [1..7] OF BOOL;
	IDX : DINT;
	XINTERNALTESTMODE : BOOL := FALSE;
	INTERNALTESTMODE : BOOL;
END_VAR
END_FUNCTION_BLOCK

(* ---- MC_SETCOORDINATETRANSFORM.pou ---- *)
FUNCTION_BLOCK MC_SETCOORDINATETRANSFORM EXTENDS L_MC4P_Template_AG_KIN
VAR_INPUT
	EXECUTE : BOOL;
	COORDTRANSFORM : MC_COORD_REF;
	COORDSYSTEM : L_MC4P_CoordSystem;
END_VAR
VAR_OUTPUT
	DONE : BOOL;
	BUSY : BOOL;
	ACTIVE : BOOL;
	COMMANDABORTED : BOOL;
	ERROR : BOOL;
	ERRORID : L_IE1P_Error;
END_VAR
VAR
	PCOORDTRAFO : POINTER TO L_MC4P_CoordTrafo;
	XEXECUTEOLD : BOOL;
	XRESETOUTPUT : BOOL;
	ISTATE : INT;
	BSTATEMACHINE : BOOL;
	PTRACKINGPARAM : POINTER TO L_MC4P_PCSTrackParam;
	COORDTRANSFFREEZE : MC_COORD_REF;
	AXPARACCESSIBLE : ARRAY [1..7] OF BOOL;
	IDX : DINT;
	XINTERNALTESTMODE : BOOL := FALSE;
	INTERNALTESTMODE : BOOL;
END_VAR
END_FUNCTION_BLOCK

(* ---- MC_SETKINTRANSFORM.pou ---- *)
FUNCTION_BLOCK MC_SETKINTRANSFORM EXTENDS L_MC4P_Template_AG_KIN
VAR_INPUT
	EXECUTE : BOOL;
	KINTRANSFORM : MC_KIN_REF;
END_VAR
VAR_OUTPUT
	DONE : BOOL;
	BUSY : BOOL;
	ACTIVE : BOOL;
	COMMANDABORTED : BOOL;
	ERROR : BOOL;
	ERRORID : L_IE1P_Error;
END_VAR
VAR
	XEXECUTEOLD : BOOL;
	XRESETOUTPUT : BOOL;
	PAXESGROUP : POINTER TO AXES_GROUP_KIN;
END_VAR
END_FUNCTION_BLOCK

(* ---- MC_TRACKCONVEYORBELT.pou ---- *)
FUNCTION_BLOCK MC_TRACKCONVEYORBELT EXTENDS L_MC4P_Template_AG_KIN_Licence
VAR_INPUT
	EXECUTE : BOOL;
	ABORT : BOOL;
	CONVEYORBELTORIGIN : ARRAY [1..6] OF LREAL;
	INITIALOBJECTPOSITION : ARRAY [1..6] OF LREAL;
	COORDSYSTEM : L_MC4P_CoordSystem;
	COORDTYPE : L_MC4P_CoordType;
	CLUTCHDISTANCE : LREAL;
	CLUTCHTIME : LREAL;
	CLUTCHTIMEABORT : LREAL;
	SETDYNPCS : BOOL := TRUE;
END_VAR
VAR_OUTPUT
	DONE : BOOL;
	BUSY : BOOL;
	ACTIVE : BOOL;
	COMMANDABORTED : BOOL;
	ERROR : BOOL;
	ERRORID : L_IE1P_Error;
	INSYNC : BOOL;
	DYNAMICPCSSET : BOOL;
END_VAR
VAR_IN_OUT
	CONVEYORBELT : AXIS_REF;
END_VAR
VAR
	TRACK : L_MC4P_TrackConveyorBelt_internal;
	CLUTCHEXTERNAL : LREAL;
	MASTERVALUESOURCE : MC_SOURCE;
END_VAR
END_FUNCTION_BLOCK

(* ---- MC_UNGROUPALLAXES.pou ---- *)
FUNCTION_BLOCK MC_UNGROUPALLAXES EXTENDS L_MC4P_Template_AG_KIN
VAR_INPUT
	EXECUTE : BOOL;
END_VAR
VAR_OUTPUT
	DONE : BOOL;
	BUSY : BOOL;
	ERROR : BOOL;
	ERRORID : L_IE1P_Error;
END_VAR
VAR
	XEXECUTEOLD : BOOL;
	XRESETOUTPUT : BOOL;
	PSDUMMY : POINTER TO STRING;
	IDX : WORD;
END_VAR
END_FUNCTION_BLOCK
